// TIA Portal V18 export
// export: Created 2026-06-09T02:47:52.5865195Z, ExportSetting WithDefaults, DisplayName Totally Integrated Automation Portal, DisplayVersion V18, DisplayName TIA Portal Openness, DisplayVersion V18, DisplayName TIA Portal Version Control Interface, DisplayVersion V18, DisplayName STEP 7 Professional, DisplayVersion V18, DisplayName STEP 7 Safety, DisplayVersion V18, DisplayName WinCC Professional, DisplayVersion V18
VAR_GLOBAL   // PLC tag table "Pakowanie"
   start_pakowaie AT %M103.0 : Bool;
   stop_pakowanie AT %M103.1 : Bool;
   cz_pojemnosciowy_pak AT %M203.0 : Bool;
   tasma_pakowanie AT %Q1.2 : Bool;
   lampa_sygnalizacyjna_pak AT %Q1.1 : Bool;
   cz_do_robota AT %Q1.3 : Bool;
END_VAR
